// TIA Portal V19 export
ORGANIZATION_BLOCK "Main"   // OB1, LAD, ProgramCycle
TITLE = "Main Program Sweep (Cycle)"
{ S7_Optimized_Access := 'TRUE' }
// h
// stored: SetENOAutomatically false
   VAR_INPUT
      Initial_Call : Bool;   // Initial call of this OB
      Remanence : Bool;   // =True, if remanent data are available
   END_VAR
   VAR_TEMP
      Start_All : Bool;
      ON : Bool;
   END_VAR
BEGIN

REGION Network 1
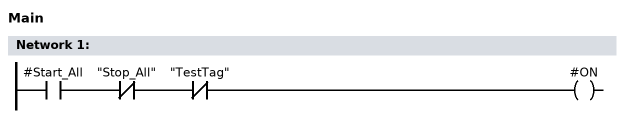
   RUNG wire#powerrail
      Contact( #Start_All )
      I_Contact( "Stop_All" )
      I_Contact( "TestTag" )
      Coil( #ON )
   END_RUNG
   // the same network as SCL:
   #ON := #Start_All AND NOT "Stop_All" AND NOT "TestTag";
END_REGION
END_ORGANIZATION_BLOCK
